// Mitsubishi GX Works2 project: z17   PLC: Q02/Q02H

PROGRAM MAIN
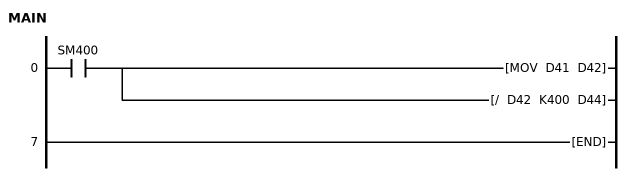
0     LD      SM400
      MOV     D41 D42
      /       D42 K400 D44
7     END
END_PROGRAM
